Universal Robots PolyScope program: Usama_Code_UR10_Maj_prog.urp

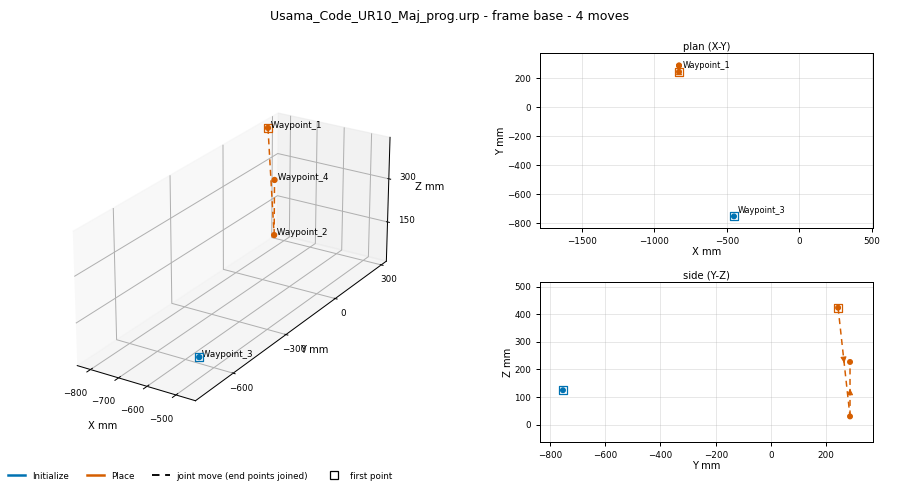
[picture p0: tool path of Usama_Code_UR10_Maj_prog.urp in frame base, 4 of 4 moves have a stored position in this frame; points joined in program order, loops and branches not executed]
Program Usama_Code_UR10_Maj_prog (installation=default directory=/programs/usbdisk/UR10_Code/UR10_Code_V3 createdIn=3.15.4.106291 lastSavedIn=3.15.4.106291 robotSerialNumber=2019300133)
Calibrated DH parameters: a=[-0.000006, -0.606471, -0.570201, -0.000053, 0.000006, 0]; d=[0.128096, 15.114888, -22.674746, 7.723348, 0.115665, 0.092162]; alpha=[1.570605, -0.005579, -0.004649, 1.571049, -1.571015, 0]; deltaTheta=[-0.00004, -0.169247, 0.199673, -0.061563, -0.000077, -0.000043]
InitVariablesNode
Robot Program (runOnlyOnce=false)
  accel := 3
  Y := 0
  SuppressedNode
    Encoder_Target := 0
  vel := 4
  Script: set_tool_voltage(24)
  Call Initialize
  SuppressedNode
    Loop While (checkContinuously=false) expression=digital_in[3] ==  True
      Call Initialize
      Call Orin_Variables
      Call Picking
      Call Place
  If digital_out[3] ==  True (checkContinuously=true)
    Call Orin_Variables
    Call Picking
    Call Place
SubProgram -> Initialize
SubProgram -> Orin_Variables
SubProgram -> Picking
SubProgram -> Place
Thread Thread_1 (runOnlyOnce=false)
  Script: socket_open("192.168.0.3", 50001, "Orin_Encoder")
  Loop Forever
    Encoder_Count := encoder_get_tick_count(0)
    Script: socket_send_line(Encoder_Count, "Orin_Encoder")
    Wait Sleep waitTime=0.1
SubProgram Initialize (keepSynchronizedWithDisk=false)
  MoveJ speed 60 deg/s, acceleration 80 deg/s^2 (useActiveTCP=true)
    Waypoint Waypoint_3: TCP in base x=-451.155 y=-752.969 z=124.774 mm, rx=-2.9238 ry=1.0806 rz=0.0968 rad; joints [49.291, -63.283, 95.687, -120.629, -94.116, -180] deg; flange x=-442.262 y=-760.597 z=301.386 mm, rx=-2.9238 ry=1.0806 rz=0.0968 rad
SubProgram Orin_Variables (keepSynchronizedWithDisk=false)
  Script: socket_open("192.168.0.3", 50002, "Orin_Y_Target")
  SuppressedNode
    Y := -0.15
  Y := socket_get_var("POS_Y", "Orin_Y_Target")
  SuppressedNode
    Script: socket_close("Orin_Y_Target")
  Y := Y / 1000
  Script: socket_open("192.168.0.3", 50000, "Orin_Encoder_Target")
  Encoder_Target := socket_get_var("Target_Encoder", "Orin_Encoder_Target")
  SuppressedNode
    Script: socket_close("Orin_Encoder_Target")
SubProgram Picking (keepSynchronizedWithDisk=false)
  SuppressedNode
    If Y > -0.2
      Halt
  Script: movej(p[-0.6, Y,  0.02, -3.02037, 0.59482, -0.03077], a  = accel, v = vel)
  Wait Condition expression=Encoder_Count ≥Encoder_Target
  SuppressedNode
    Halt
  URCap Conveyor Tracking (Conveyor Tracking, Universal Robots)
    Script: current_pose= get_target_tcp_pose()
    new_pose := p[current_pose[0], current_pose[1], current_pose[2] - 0.017, current_pose[3], current_pose[4], current_pose[5]]
    Script: movej(new_pose, a= accel, v = vel)
    SuppressedNode
      URCap SMC Vacuum Gripper Unit (SMC Vacuum Gripper Unit, SMC Corporation.) dataModel(adsorbLevel=-60, vacuumLevelCheckTime=1000, blowOffTime=100, blowOffTimeCommissioning=100, workpieceWeight=0.05, adsorbNodeFunction=true, checkWaitVacuumLevel=true)
  SuppressedNode
    If Encoder_Count == Encoder_Target
      URCap Conveyor Tracking (Conveyor Tracking, Universal Robots)
        Script: current_pose= get_target_tcp_pose()
        new_pose := p[current_pose[0], current_pose[1], current_pose[2] - 0.017, current_pose[3], current_pose[4], current_pose[5]]
        Script: movej(new_pose, a= accel, v = vel)
        URCap SMC Vacuum Gripper Unit (SMC Vacuum Gripper Unit, SMC Corporation.) dataModel(adsorbLevel=-60, vacuumLevelCheckTime=1000, blowOffTime=100, blowOffTimeCommissioning=100, workpieceWeight=0.05, adsorbNodeFunction=true, checkWaitVacuumLevel=true)
  SuppressedNode
    Loop While (checkContinuously=false) expression=Encoder_Count == Encoder_Target
      URCap Conveyor Tracking (Conveyor Tracking, Universal Robots)
        Script: current_pose= get_target_tcp_pose()
        new_pose := p[current_pose[0], current_pose[1], current_pose[2] - 0.017, current_pose[3], current_pose[4], current_pose[5]]
        Script: movej(new_pose, a= accel, v = vel)
        URCap SMC Vacuum Gripper Unit (SMC Vacuum Gripper Unit, SMC Corporation.) dataModel(adsorbLevel=-60, vacuumLevelCheckTime=1000, blowOffTime=100, blowOffTimeCommissioning=100, workpieceWeight=0.05, adsorbNodeFunction=true, checkWaitVacuumLevel=true)
SubProgram Place (keepSynchronizedWithDisk=false)
  MoveJ speed 60 deg/s, acceleration 80 deg/s^2 (useActiveTCP=true)
    Waypoint Waypoint_1: TCP in base x=-829.878 y=242.735 z=423.377 mm, rx=-1.6327 ry=2.616 rz=0.05 rad; joints [-26.258, -72.408, 76.794, -92.44, -94.096, -179.916] deg; flange x=-835.472 y=232.478 z=599.991 mm, rx=-1.6327 ry=2.616 rz=0.05 rad
    Waypoint Waypoint_2: TCP in base x=-829.88 y=285.88 z=29.908 mm, rx=-1.5727 ry=2.6531 rz=0.0521 rad; joints [-28.783, -58.173, 99.103, -129.16, -94.113, -180] deg; flange x=-835.495 y=275.615 z=206.521 mm, rx=-1.5727 ry=2.6531 rz=0.0521 rad
    SuppressedNode
      URCap SMC Vacuum Gripper Unit (SMC Vacuum Gripper Unit, SMC Corporation.) dataModel(adsorbLevel=-60, vacuumLevelCheckTime=1000, blowOffTime=100, blowOffTimeCommissioning=100, adsorbNodeFunction=false, checkWaitVacuumLevel=false)
    Waypoint Waypoint_4: TCP in base x=-829.858 y=285.966 z=227.061 mm, rx=-1.5742 ry=2.6522 rz=0.0522 rad; joints [-28.803, -67.464, 90.389, -111.155, -94.115, -180] deg; flange x=-835.467 y=275.679 z=403.673 mm, rx=-1.5742 ry=2.6522 rz=0.0522 rad
    Script: set_digital_out(3,  False )
